TYPE Orient_Outputs_typ:
STRUCT
	BallClampOpen AT %Q*: BOOL;
	BallClampClose AT %Q*: BOOL;
	LoadBall AT %Q*: BOOL;
END_STRUCT
END_TYPE

(* stored: Version 1.1.0.1, ProductVersion 3.1.4024.12
   DUT Orient_Outputs_typ: Id {9c611e32-5366-0f50-34dd-2ab9b34151b3} *)
